# B&R Automation Studio project Projekt_v_1_0
Automation Studio 4.3.6.57 SP; technology packages: mappView 5.3.2

## Configuration Config1

CPU PC_any, AutomationRuntime E4.34, Build 4.1.2, Vc V4.34.3

CPU X20CP1382, AutomationRuntime E4.34, Build 4.1.2, Vc V4.34.3

### Task classes (Cpu.sw)
```
Cyclic#3:
  Program <- VisuDemoWall.Program.prg
Binaries: TCData, udbdef, mvLoader, sysconf, ashwac, arconfig, asfw, User, ashwd, iomap, Role, OpcUaMap
Libraries: fileio, astime, runtime, asieccon
```

### Task classes (Cpu.sw)
```

```

### Hardware
```
PC : PC_any v1.1.0.0 (OrderNumber=PC)
  ConfigurationID = Projekt_v_1_0_Config1
  ActivateOpcUa = 1
  OpcUaInformationModels_PV_Version = 1
```

## Configuration Panel

CPU 5PPC2100.BY44-000, AutomationRuntime I4.33, Build 4.1.2

### Task classes (Cpu.sw)
```
Cyclic#5:
  Program <- VisuDemoWall.Program.prg
Binaries: udbdef, mvLoader, TCLang, TCData, ashwac, Role, ashwd, arconfig, iomap, OpcUaMap, asfw, sysconf, TC, User
Libraries: asieccon, astime, runtime, fileio
```

### Hardware
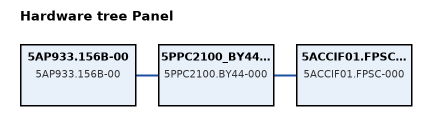
```
5ACCIF01.FPSC-000 : 5ACCIF01.FPSC-000 v1.2.1.0  [SL -> 5PPC2100_BY44_000.SL1]
5AP933.156B-00 : 5AP933.156B-00 v1.4.0.1
5PPC2100_BY44_000 : 5PPC2100.BY44-000 v1.2.4.0  [SY -> 5AP933.156B-00.SY1]
  Connector IF3:
    ActivateDevice = 1
  Connector IF4:
    ActivateDevice = 1
  AutomationRuntime = AR010
  ConfigurationID = Projekt_v_1_0_Panel
  StartMode = 0
  ActivateOpcUa = 1
  OpcUa_AuthenticationSecurityPolicy_EnableNone = 1
  OpcUa_AuthenticationSecurityPolicy_EnableBasic128Rsa15 = 1
  OpcUaInformationModels_PV_Version = 1
```

## Logical view

Binary libraries used (declarations not repeated): operator, runtime, astime, AsIecCon

### Package Logical/Libraries - Global libraries

- Visualisation Logical/VisuDemoWall (not shown)

- Visualisation Logical/mappView (not shown)

### Global.typ - not listed in the package file held
```iecst
TYPE
<<<<<<< HEAD

=======
	TypDanych : 	STRUCT
		lol : USINT;
		Lol1 : USINT;
	END_STRUCT;
>>>>>>> Kamil
END_TYPE
```

### Global.var - not listed in the package file held
```iecst
VAR
	ZmiennaKamila : USINT;
END_VAR
```
